// TIA Portal V18 export
DATA_BLOCK "DB_LHTTPControl"   // DB7
{ S7_Optimized_Access := 'TRUE' }
// stored: MemoryReserve 100
   VAR
      postCommand : Bool;
      extractedDataName : String;
      extractedDataDescription : String;
      extractedDataMessage : String;
      Body : String := '{"keyID":"KEY15"}';
      geturl : String;
      PostOrPut : USInt;
   END_VAR
BEGIN
END_DATA_BLOCK
